FUNCTION_BLOCK FB_ScaleOut_1
VAR_INPUT
	inputForScaling : REAL;
	inMin : REAL;
	inMax : REAL;
	outMin : REAL;
	outMax : REAL;
	ctrlCycletime : TIME;
	taskCycletime : TIME;
END_VAR
VAR_OUTPUT
	scaledOutput : real;
END_VAR
VAR
	fbScale : FB_CTRL_SCALE;
	stParamsForScaling : ST_CTRL_SCALE_PARAMS;
	
END_VAR

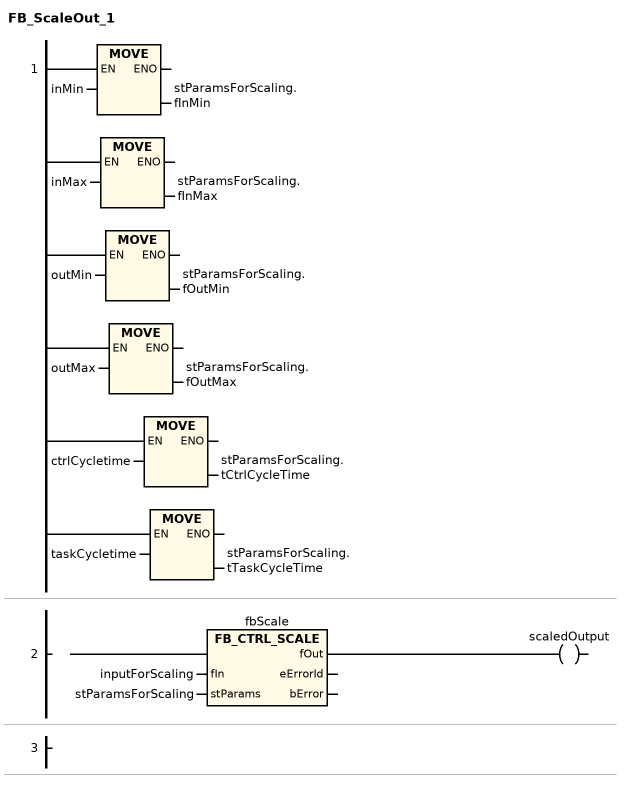
// NETWORK 1
stParamsForScaling.fInMin := inMin;
stParamsForScaling.fInMax := inMax;
stParamsForScaling.fOutMin := outMin;
stParamsForScaling.fOutMax := outMax;
stParamsForScaling.tCtrlCycleTime := ctrlCycletime;
stParamsForScaling.tTaskCycleTime := taskCycletime;

// NETWORK 2
fbScale(fIn := inputForScaling, stParams := stParamsForScaling); // FB_CTRL_SCALE
scaledOutput := fbScale.fOut;

// NETWORK 3

END_FUNCTION_BLOCK

(* stored: Version 1.1.0.1, ProductVersion 3.1.4024.13
   POU FB_ScaleOut_1: Id {5573dff7-e7a5-46b9-adaf-a81cb9ea2a13}, SpecialFunc None *)
